(* Logix 5000 project; controller LeakTestAuto vendor 1 type 14 code 226 rev 37.11; software revision 37.01; part 5 of 13 *)
(* tags used below, declared in another part *)
   AOI_Barcode_Comms : AOI_CommStatus;
   AOI_CTS1 : AOI_CTS_INSTRUMENT;
   AOI_CTS1_Comms : AOI_CommStatus;
   AOI_CTS2 : AOI_CTS_INSTRUMENT;
   AOI_CTS2_Comms : AOI_CommStatus;
   AOI_GetShift : AOI_GetShift;
   AOI_RFID_Comms : AOI_CommStatus;
   AOI_Robot_Comms : AOI_CommStatus;
   AOI_RobotPos : AOI_RobotPositions;
   AOI_SeqSteps : AOI_StandardSeqSteps;
   BarcodeScanner : udt_OutputStructure;
   CapActuators_Seq : udt_SequenceStructure_X64;
   CapCTS_Seq : udt_SequenceStructure_X64;
   CapCylinders_Seq : udt_SequenceStructure_X64;
   CapFail_Seq : udt_SequenceStructure_X64;
   CapPass_Seq : udt_SequenceStructure_X64;
   CapRobot_Seq : udt_SequenceStructure_X64;
   CapShuffle_Seq : udt_SequenceStructure_X64;
   Conveyor : udt_OutputStructure;
   ConveyorHomeCounter : COUNTER;
   DryCycle_N1Ready : BOOL;
   DryCycle_N2Ready : BOOL;
   HMI_CloseDisplay : DINT;
   HomingClearNestsBypass : BOOL;
   LastShiftNumber : DINT;
   LeakTester1 : udt_OutputStructure;
   LeakTester2 : udt_OutputStructure;
   Mode_CapActuators : BOOL;
   Mode_CapCTS : BOOL;
   Mode_CapCylinders : BOOL;
   Mode_CapFail : BOOL;
   Mode_CapPass : BOOL;
   Mode_CapRobot : BOOL;
   Mode_CapShuffle : BOOL;
   Nest1Cylinder : udt_OutputStructure;
   Nest2Cylinder : udt_OutputStructure;
   ONS_CapActuators : BOOL;
   ONS_CapCTS : BOOL;
   ONS_CapCylinders : BOOL;
   ONS_CapFail : BOOL;
   ONS_CapPass : BOOL;
   ONS_CapRobot : BOOL;
   ONS_CapShuffle : BOOL;
   ONS_CycleStop : BOOL;
   ONS_ManuMode : BOOL;
   OP220 : udt_Mode;
   OP220_PartToPartCycleTMR : TIMER;
   OP220_Seq : udt_SequenceStructure_X64;
   RFIDScanner : udt_OutputStructure;
   Robot : udt_OutputStructure;
   RobotGripper : udt_OutputStructure;
   RobotInputs : udt_EpsonInputs;
   RobotOutputs : udt_EpsonOutputs;
   ShiftTimes : SINT[24];
   TON_HMICloseDisplayDelay : TIMER;
   ConveyorPurgeCounter : DINT;   // Outfeed Coveyor Purge Counter
   DateString : String20;
   DateTimeString : String20;
   HMI_PurgeCycleSP : DINT;   // HMI Purge Cycles Setpoint
   I_OP220_N3_CONVEYOR_CLEAT : ALIAS FOR Local:3:I.Pt13.Data;
   I_OP220_N3_CONVEYOR_LOAD : ALIAS FOR Local:3:I.Pt12.Data;
   I_OP220_N3_CONVEYOR_UNLOAD : ALIAS FOR Local:3:I.Pt14.Data;
   I_OP220_N3_DUT_PRE_NEST_0 : ALIAS FOR Local:3:I.Pt00.Data;
   I_OP220_N3_DUT_PRE_NEST_1 : ALIAS FOR Local:3:I.Pt01.Data;
   I_OP220_N3_DUT_PRE_NEST_2 : ALIAS FOR Local:3:I.Pt02.Data;
   I_OP220_N3_MAIN_AIR_OK : ALIAS FOR Local:3:I.Pt07.Data;
   I_OP220_N3_NEST1_EXTEND : ALIAS FOR Local:3:I.Pt04.Data;
   I_OP220_N3_NEST1_HOME : ALIAS FOR Local:3:I.Pt03.Data;
   I_OP220_N3_NEST2_EXTEND : ALIAS FOR Local:3:I.Pt06.Data;
   I_OP220_N3_NEST2_HOME : ALIAS FOR Local:3:I.Pt05.Data;
   I_OP220_N3_REJECT_BIN_OK : ALIAS FOR Local:3:I.Pt09.Data;
   IOCounterHasRef : BOOL;
   IOTriggerCounts : UDINT[128];
   James_Dint : DINT;   // James Test Word
   LastPLCEdit : String20;
   LastPLCEditHistory : String20[20];
   O_OP220_N5_EN_LT_BU : ALIAS FOR Local:5:O.Pt03.Data;
   O_OP220_N5_EN_LT_GN : ALIAS FOR Local:5:O.Pt00.Data;
   O_OP220_N5_EN_LT_RD : ALIAS FOR Local:5:O.Pt02.Data;
   O_OP220_N5_EN_LT_YE : ALIAS FOR Local:5:O.Pt01.Data;
   OP220_ConsumedFromMain_PurgeModeEn : BOOL;
   OP220_Power : BOOL;
   PLC : AOI_PLC;
   Purge_Count_DN : BOOL;   // Purge Counter Completed
   ShiftChange : BOOL;
   ShiftNumber : SINT;
   TimeString : String20;
   TON_PLC_BootUp : TIMER;
(* MainProgram, continued *)

ROUTINE AManualDebug   (* ladder *)
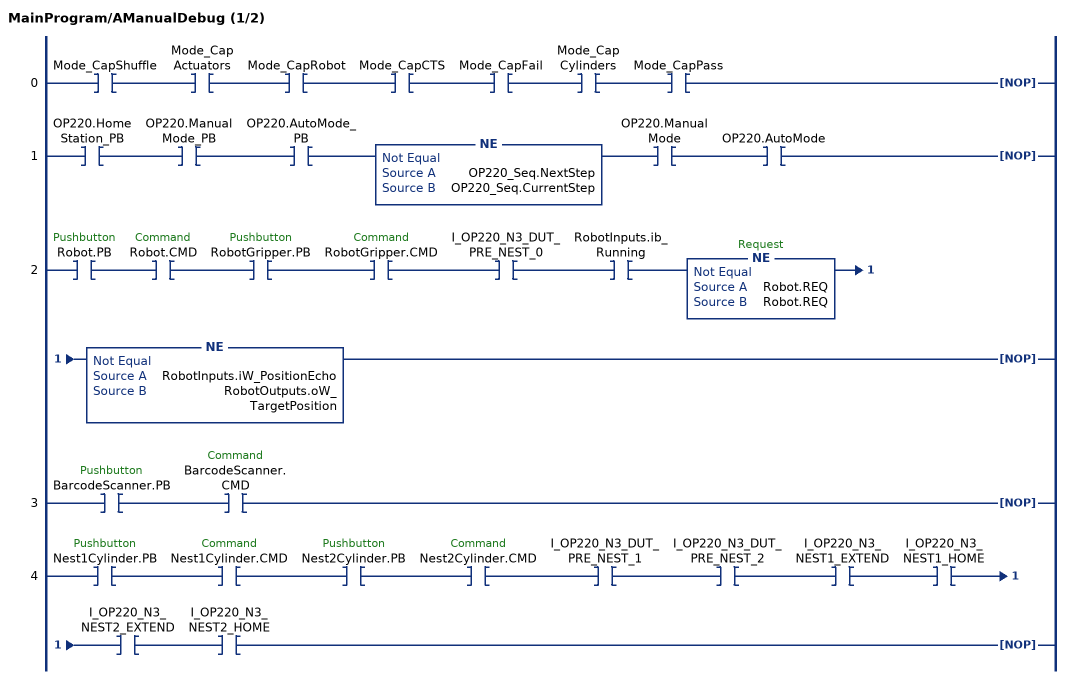
   0: XIC(Mode_CapShuffle)XIC(Mode_CapActuators)XIC(Mode_CapRobot)XIC(Mode_CapCTS)XIC(Mode_CapFail)XIC(Mode_CapCylinders)XIC(Mode_CapPass)NOP();
   1: XIC(OP220.HomeStation_PB)XIC(OP220.ManualMode_PB)XIC(OP220.AutoMode_PB)NE(OP220_Seq.NextStep,OP220_Seq.CurrentStep)XIC(OP220.ManualMode)XIC(OP220.AutoMode)NOP();
   2: XIC(Robot.PB)XIC(Robot.CMD)XIC(RobotGripper.PB)XIC(RobotGripper.CMD)XIC(I_OP220_N3_DUT_PRE_NEST_0)XIC(RobotInputs.ib_Running)NE(Robot.REQ,Robot.REQ)NE(RobotInputs.iW_PositionEcho,RobotOutputs.oW_TargetPosition)NOP();
   3: XIC(BarcodeScanner.PB)XIC(BarcodeScanner.CMD)NOP();
   4: XIC(Nest1Cylinder.PB)XIC(Nest1Cylinder.CMD)XIC(Nest2Cylinder.PB)XIC(Nest2Cylinder.CMD)XIC(I_OP220_N3_DUT_PRE_NEST_1)XIC(I_OP220_N3_DUT_PRE_NEST_2)XIC(I_OP220_N3_NEST1_EXTEND)XIC(I_OP220_N3_NEST1_HOME)XIC(I_OP220_N3_NEST2_EXTEND)XIC(I_OP220_N3_NEST2_HOME)NOP();
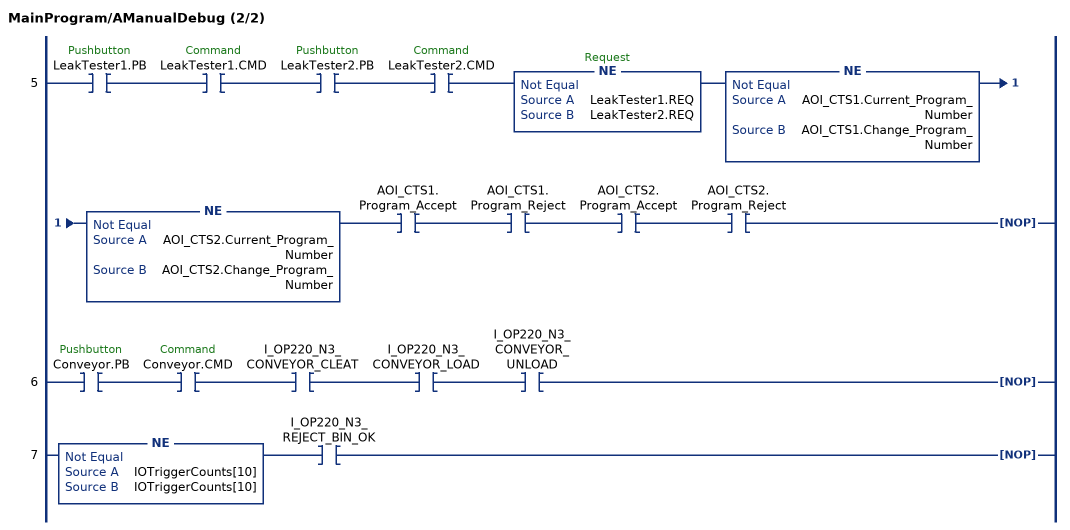
   5: XIC(LeakTester1.PB)XIC(LeakTester1.CMD)XIC(LeakTester2.PB)XIC(LeakTester2.CMD)NE(LeakTester1.REQ,LeakTester2.REQ)NE(AOI_CTS1.Current_Program_Number,AOI_CTS1.Change_Program_Number)NE(AOI_CTS2.Current_Program_Number,AOI_CTS2.Change_Program_Number)XIC(AOI_CTS1.Program_Accept)XIC(AOI_CTS1.Program_Reject)XIC(AOI_CTS2.Program_Accept)XIC(AOI_CTS2.Program_Reject)NOP();
   6: XIC(Conveyor.PB)XIC(Conveyor.CMD)XIC(I_OP220_N3_CONVEYOR_CLEAT)XIC(I_OP220_N3_CONVEYOR_LOAD)XIC(I_OP220_N3_CONVEYOR_UNLOAD)NOP();
   7: NE(IOTriggerCounts[10],IOTriggerCounts[10])XIC(I_OP220_N3_REJECT_BIN_OK)NOP();
END_ROUTINE

ROUTINE MainRoutine   (* ladder *)
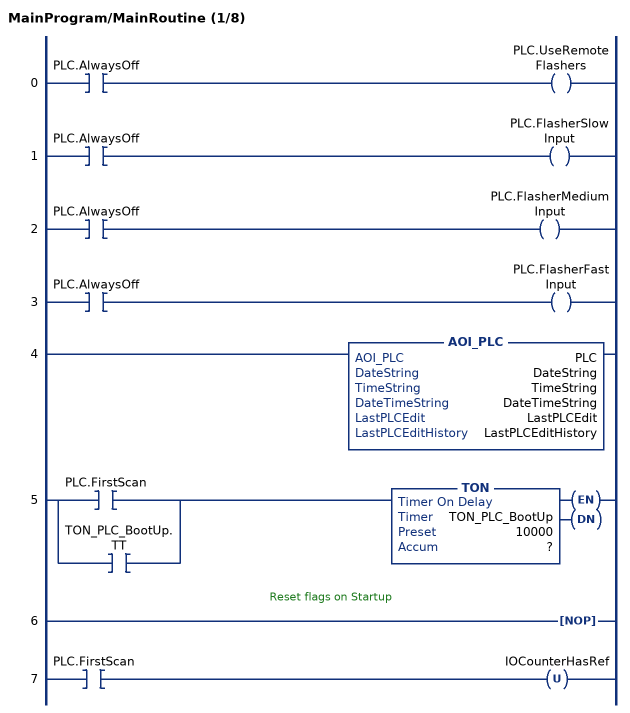
   0: XIC(PLC.AlwaysOff)OTE(PLC.UseRemoteFlashers);
   1: XIC(PLC.AlwaysOff)OTE(PLC.FlasherSlowInput);
   2: XIC(PLC.AlwaysOff)OTE(PLC.FlasherMediumInput);
   3: XIC(PLC.AlwaysOff)OTE(PLC.FlasherFastInput);
   4: AOI_PLC(PLC,DateString,TimeString,DateTimeString,LastPLCEdit,LastPLCEditHistory);
   5: [XIC(PLC.FirstScan) ,XIC(TON_PLC_BootUp.TT) ]TON(TON_PLC_BootUp,?,?);
   // Reset flags on Startup
   6: NOP();
   7: XIC(PLC.FirstScan)OTU(IOCounterHasRef);
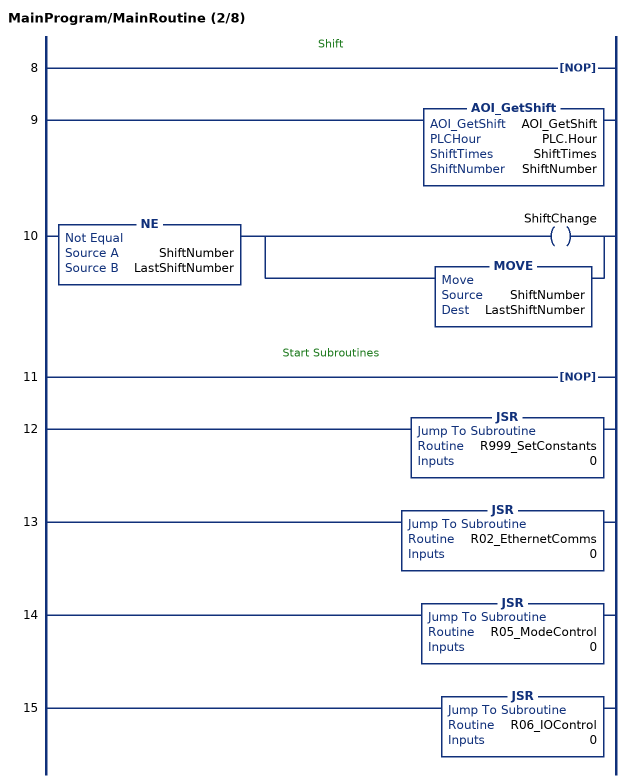
   // Shift
   8: NOP();
   9: AOI_GetShift(AOI_GetShift,PLC.Hour,ShiftTimes,ShiftNumber);
   10: NE(ShiftNumber,LastShiftNumber)[OTE(ShiftChange) ,MOVE(ShiftNumber,LastShiftNumber) ];
   // Start Subroutines
   11: NOP();
   12: JSR(R999_SetConstants,0);
   13: JSR(R02_EthernetComms,0);
   14: JSR(R05_ModeControl,0);
   15: JSR(R06_IOControl,0);
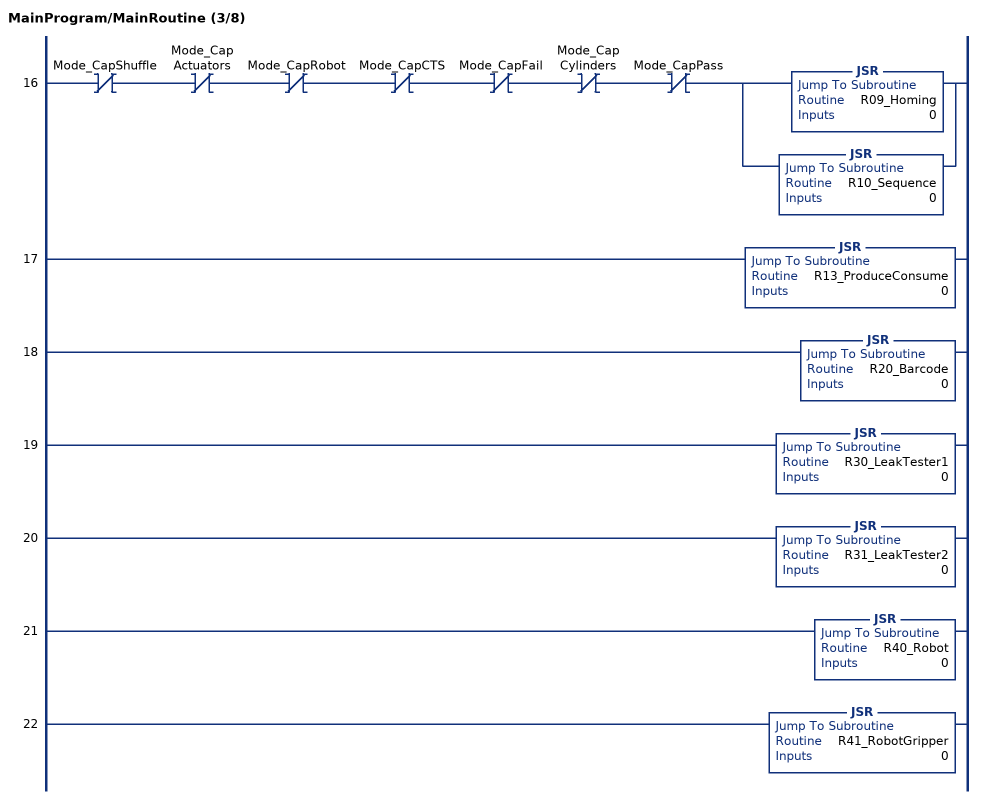
   16: XIO(Mode_CapShuffle)XIO(Mode_CapActuators)XIO(Mode_CapRobot)XIO(Mode_CapCTS)XIO(Mode_CapFail)XIO(Mode_CapCylinders)XIO(Mode_CapPass)[JSR(R09_Homing,0) ,JSR(R10_Sequence,0) ];
   17: JSR(R13_ProduceConsume,0);
   18: JSR(R20_Barcode,0);
   19: JSR(R30_LeakTester1,0);
   20: JSR(R31_LeakTester2,0);
   21: JSR(R40_Robot,0);
   22: JSR(R41_RobotGripper,0);
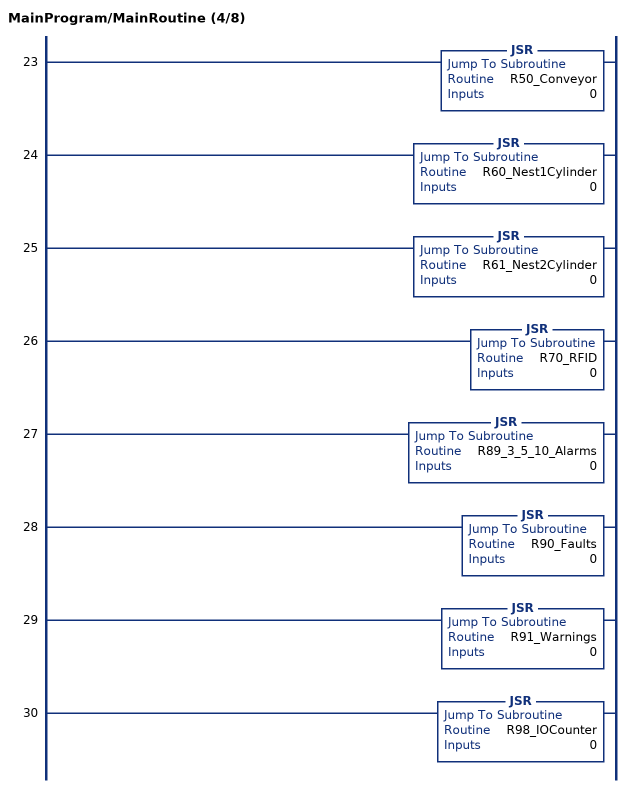
   23: JSR(R50_Conveyor,0);
   24: JSR(R60_Nest1Cylinder,0);
   25: JSR(R61_Nest2Cylinder,0);
   26: JSR(R70_RFID,0);
   27: JSR(R89_3_5_10_Alarms,0);
   28: JSR(R90_Faults,0);
   29: JSR(R91_Warnings,0);
   30: JSR(R98_IOCounter,0);
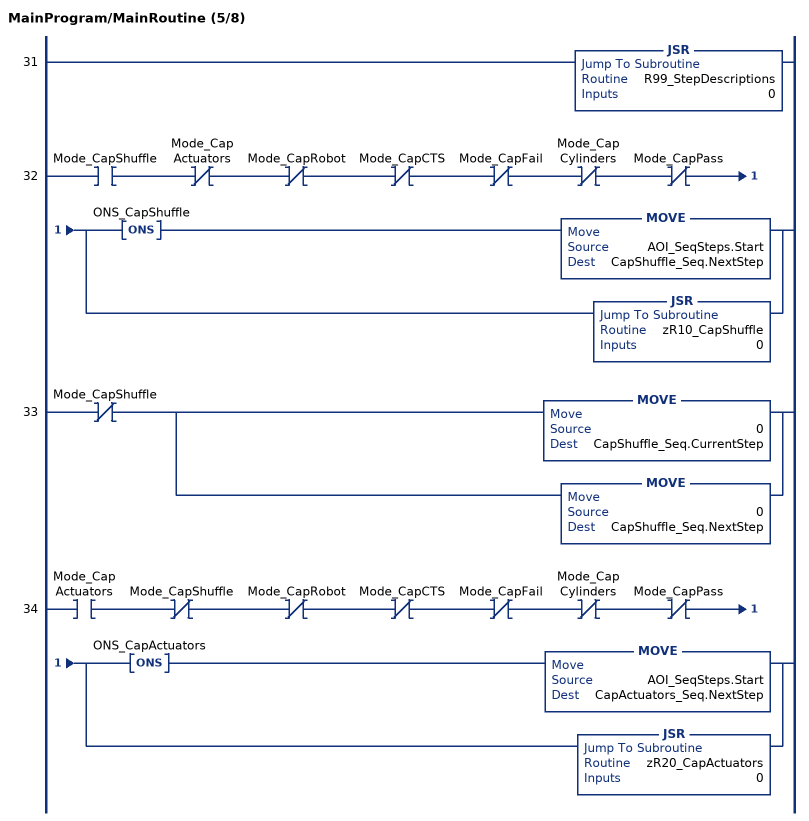
   31: JSR(R99_StepDescriptions,0);
   32: XIC(Mode_CapShuffle)XIO(Mode_CapActuators)XIO(Mode_CapRobot)XIO(Mode_CapCTS)XIO(Mode_CapFail)XIO(Mode_CapCylinders)XIO(Mode_CapPass)[ONS(ONS_CapShuffle) MOVE(AOI_SeqSteps.Start,CapShuffle_Seq.NextStep) ,JSR(zR10_CapShuffle,0) ];
   33: XIO(Mode_CapShuffle)[MOVE(0,CapShuffle_Seq.CurrentStep) ,MOVE(0,CapShuffle_Seq.NextStep) ];
   34: XIC(Mode_CapActuators)XIO(Mode_CapShuffle)XIO(Mode_CapRobot)XIO(Mode_CapCTS)XIO(Mode_CapFail)XIO(Mode_CapCylinders)XIO(Mode_CapPass)[ONS(ONS_CapActuators) MOVE(AOI_SeqSteps.Start,CapActuators_Seq.NextStep) ,JSR(zR20_CapActuators,0) ];
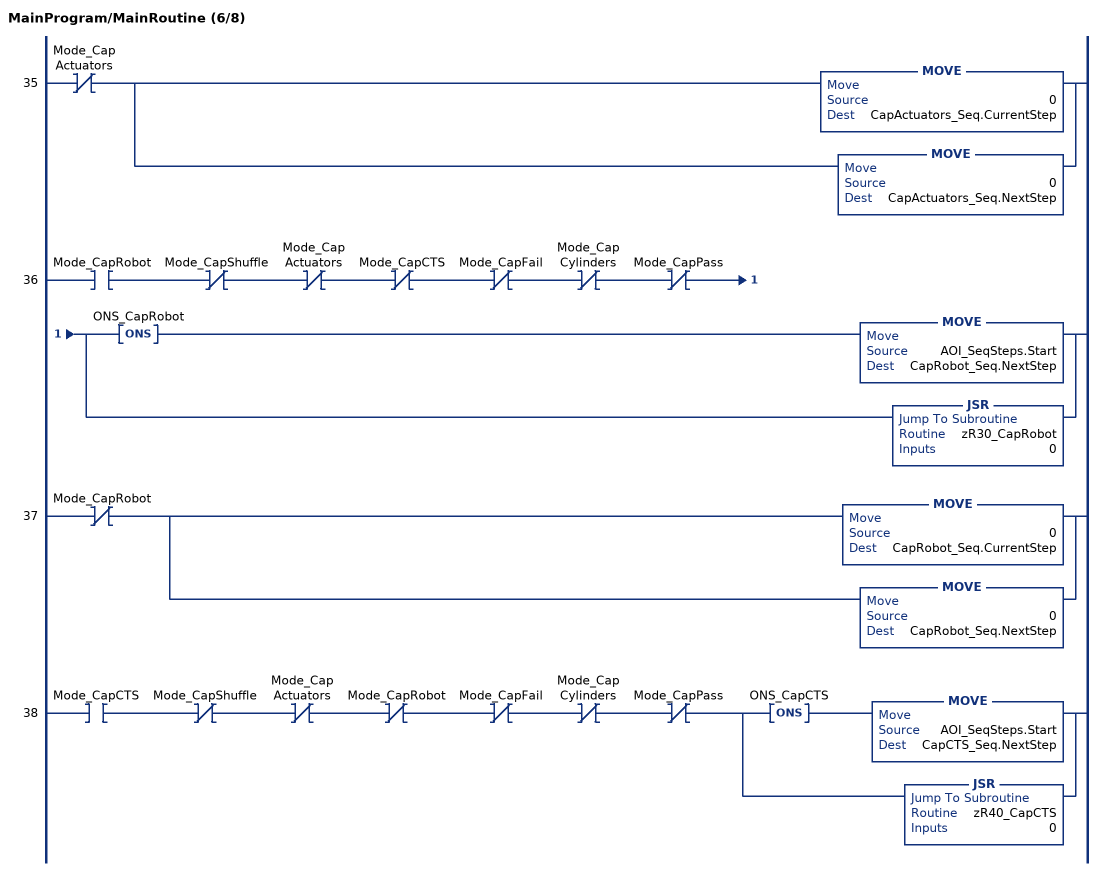
   35: XIO(Mode_CapActuators)[MOVE(0,CapActuators_Seq.CurrentStep) ,MOVE(0,CapActuators_Seq.NextStep) ];
   36: XIC(Mode_CapRobot)XIO(Mode_CapShuffle)XIO(Mode_CapActuators)XIO(Mode_CapCTS)XIO(Mode_CapFail)XIO(Mode_CapCylinders)XIO(Mode_CapPass)[ONS(ONS_CapRobot) MOVE(AOI_SeqSteps.Start,CapRobot_Seq.NextStep) ,JSR(zR30_CapRobot,0) ];
   37: XIO(Mode_CapRobot)[MOVE(0,CapRobot_Seq.CurrentStep) ,MOVE(0,CapRobot_Seq.NextStep) ];
   38: XIC(Mode_CapCTS)XIO(Mode_CapShuffle)XIO(Mode_CapActuators)XIO(Mode_CapRobot)XIO(Mode_CapFail)XIO(Mode_CapCylinders)XIO(Mode_CapPass)[ONS(ONS_CapCTS) MOVE(AOI_SeqSteps.Start,CapCTS_Seq.NextStep) ,JSR(zR40_CapCTS,0) ];
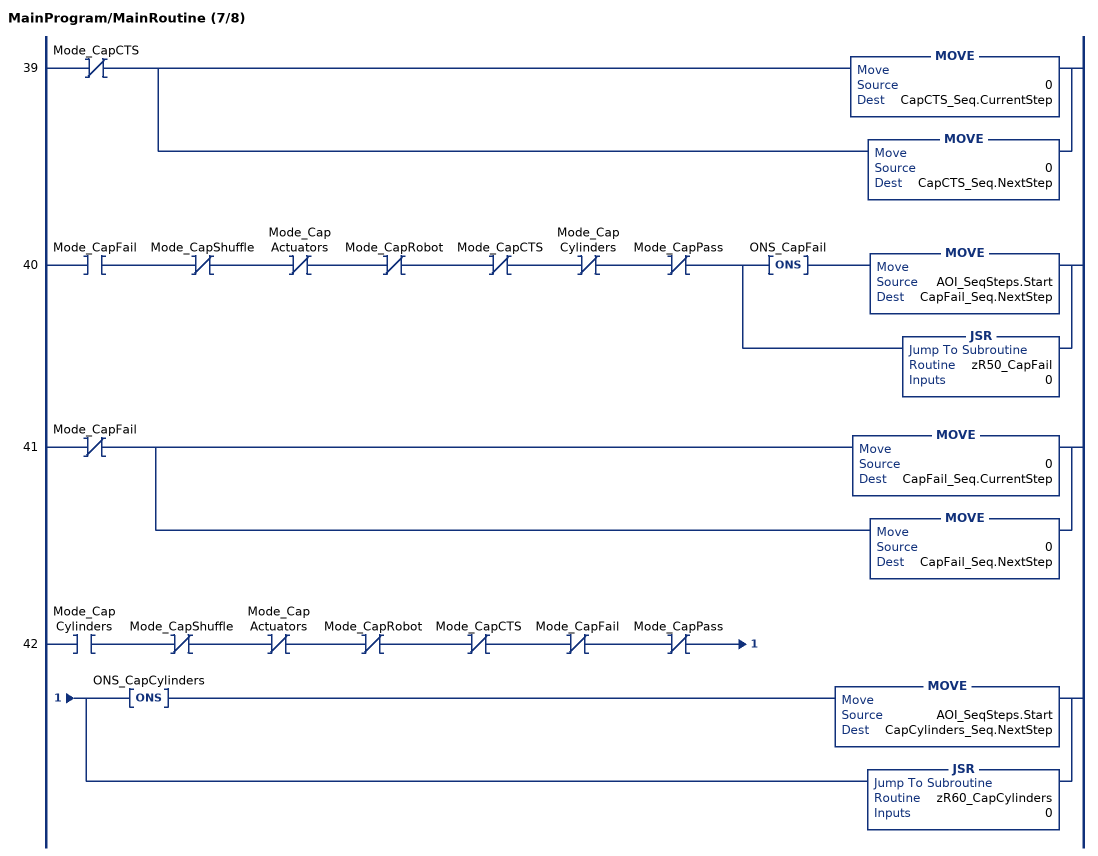
   39: XIO(Mode_CapCTS)[MOVE(0,CapCTS_Seq.CurrentStep) ,MOVE(0,CapCTS_Seq.NextStep) ];
   40: XIC(Mode_CapFail)XIO(Mode_CapShuffle)XIO(Mode_CapActuators)XIO(Mode_CapRobot)XIO(Mode_CapCTS)XIO(Mode_CapCylinders)XIO(Mode_CapPass)[ONS(ONS_CapFail) MOVE(AOI_SeqSteps.Start,CapFail_Seq.NextStep) ,JSR(zR50_CapFail,0) ];
   41: XIO(Mode_CapFail)[MOVE(0,CapFail_Seq.CurrentStep) ,MOVE(0,CapFail_Seq.NextStep) ];
   42: XIC(Mode_CapCylinders)XIO(Mode_CapShuffle)XIO(Mode_CapActuators)XIO(Mode_CapRobot)XIO(Mode_CapCTS)XIO(Mode_CapFail)XIO(Mode_CapPass)[ONS(ONS_CapCylinders) MOVE(AOI_SeqSteps.Start,CapCylinders_Seq.NextStep) ,JSR(zR60_CapCylinders,0) ];
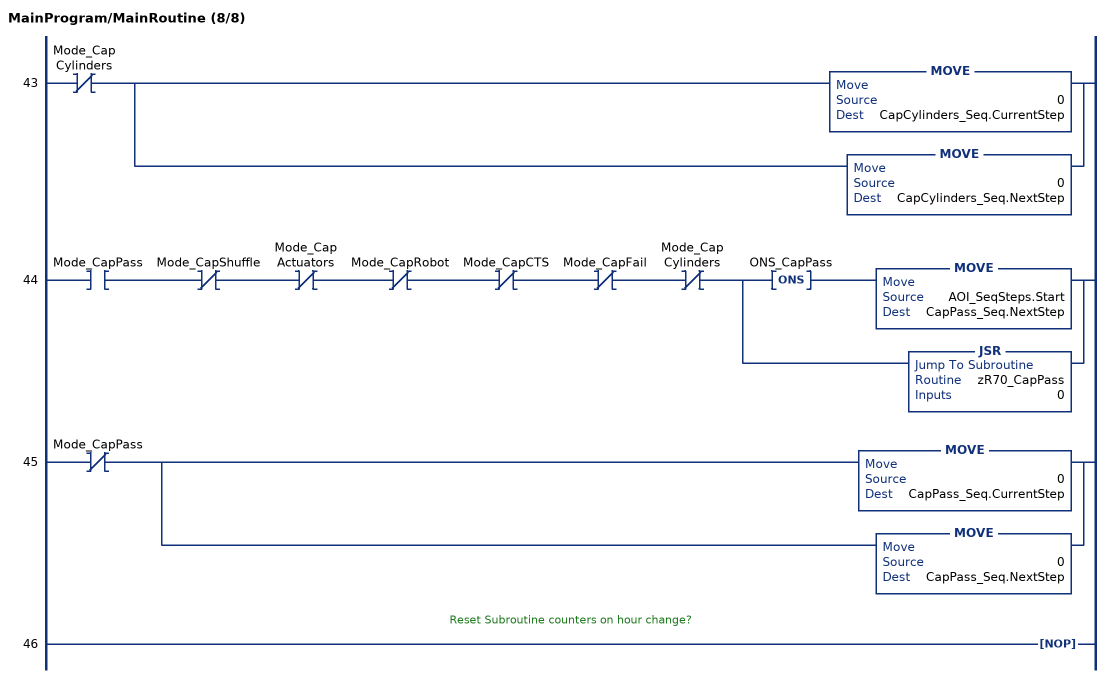
   43: XIO(Mode_CapCylinders)[MOVE(0,CapCylinders_Seq.CurrentStep) ,MOVE(0,CapCylinders_Seq.NextStep) ];
   44: XIC(Mode_CapPass)XIO(Mode_CapShuffle)XIO(Mode_CapActuators)XIO(Mode_CapRobot)XIO(Mode_CapCTS)XIO(Mode_CapFail)XIO(Mode_CapCylinders)[ONS(ONS_CapPass) MOVE(AOI_SeqSteps.Start,CapPass_Seq.NextStep) ,JSR(zR70_CapPass,0) ];
   45: XIO(Mode_CapPass)[MOVE(0,CapPass_Seq.CurrentStep) ,MOVE(0,CapPass_Seq.NextStep) ];
   // Reset Subroutine counters on hour change?
   46: NOP();
END_ROUTINE

ROUTINE R02_EthernetComms   (* ladder *)
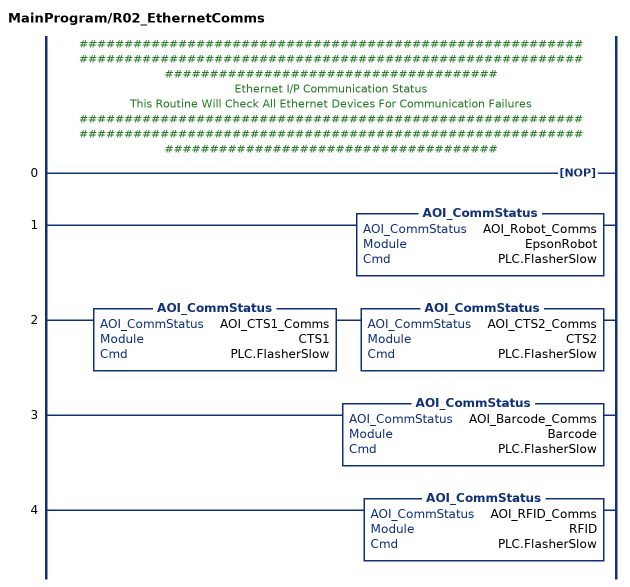
   // #####################################################################################################################################################
   // Ethernet I/P Communication Status
   // This Routine Will Check All Ethernet Devices For Communication Failures
   // #####################################################################################################################################################
   0: NOP();
   1: AOI_CommStatus(AOI_Robot_Comms,EpsonRobot,PLC.FlasherSlow);
   2: AOI_CommStatus(AOI_CTS1_Comms,CTS1,PLC.FlasherSlow)AOI_CommStatus(AOI_CTS2_Comms,CTS2,PLC.FlasherSlow);
   3: AOI_CommStatus(AOI_Barcode_Comms,Barcode,PLC.FlasherSlow);
   4: AOI_CommStatus(AOI_RFID_Comms,RFID,PLC.FlasherSlow);
END_ROUTINE

ROUTINE R05_ModeControl   (* ladder *)
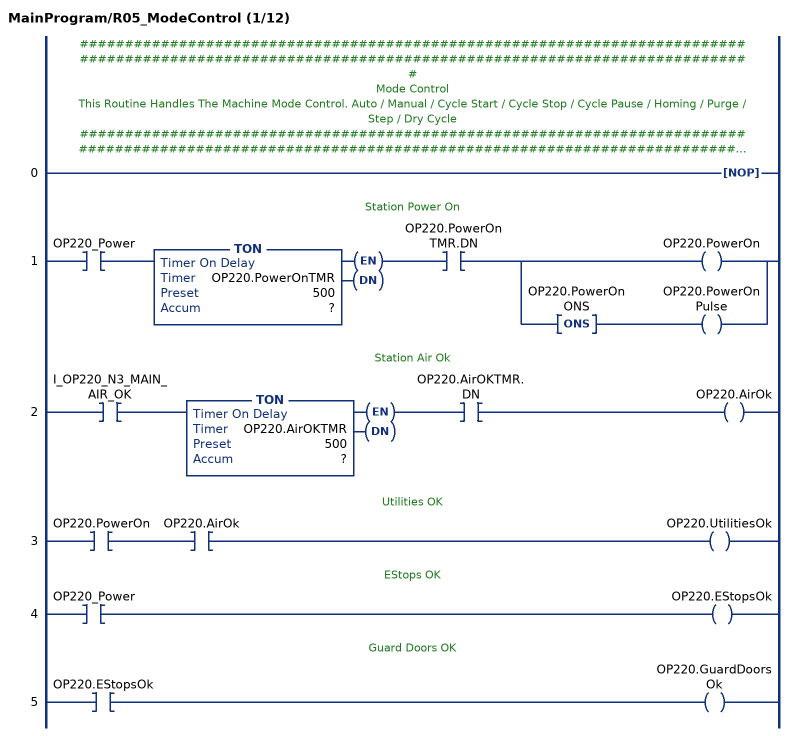
   // #####################################################################################################################################################
   // Mode Control
   // This Routine Handles The Machine Mode Control. Auto / Manual / Cycle Start / Cycle Stop / Cycle Pause / Homing / Purge / Step / Dry Cycle
   // #####################################################################################################################################################
   0: NOP();
   // Station Power On
   1: XIC(OP220_Power)TON(OP220.PowerOnTMR,?,?)XIC(OP220.PowerOnTMR.DN)[OTE(OP220.PowerOn) ,ONS(OP220.PowerOnONS) OTE(OP220.PowerOnPulse) ];
   // Station Air Ok
   2: XIC(I_OP220_N3_MAIN_AIR_OK)TON(OP220.AirOKTMR,?,?)XIC(OP220.AirOKTMR.DN)OTE(OP220.AirOk);
   // Utilities OK
   3: XIC(OP220.PowerOn)XIC(OP220.AirOk)OTE(OP220.UtilitiesOk);
   // EStops OK
   4: XIC(OP220_Power)OTE(OP220.EStopsOk);
   // Guard Doors OK
   5: XIC(OP220.EStopsOk)OTE(OP220.GuardDoorsOk);
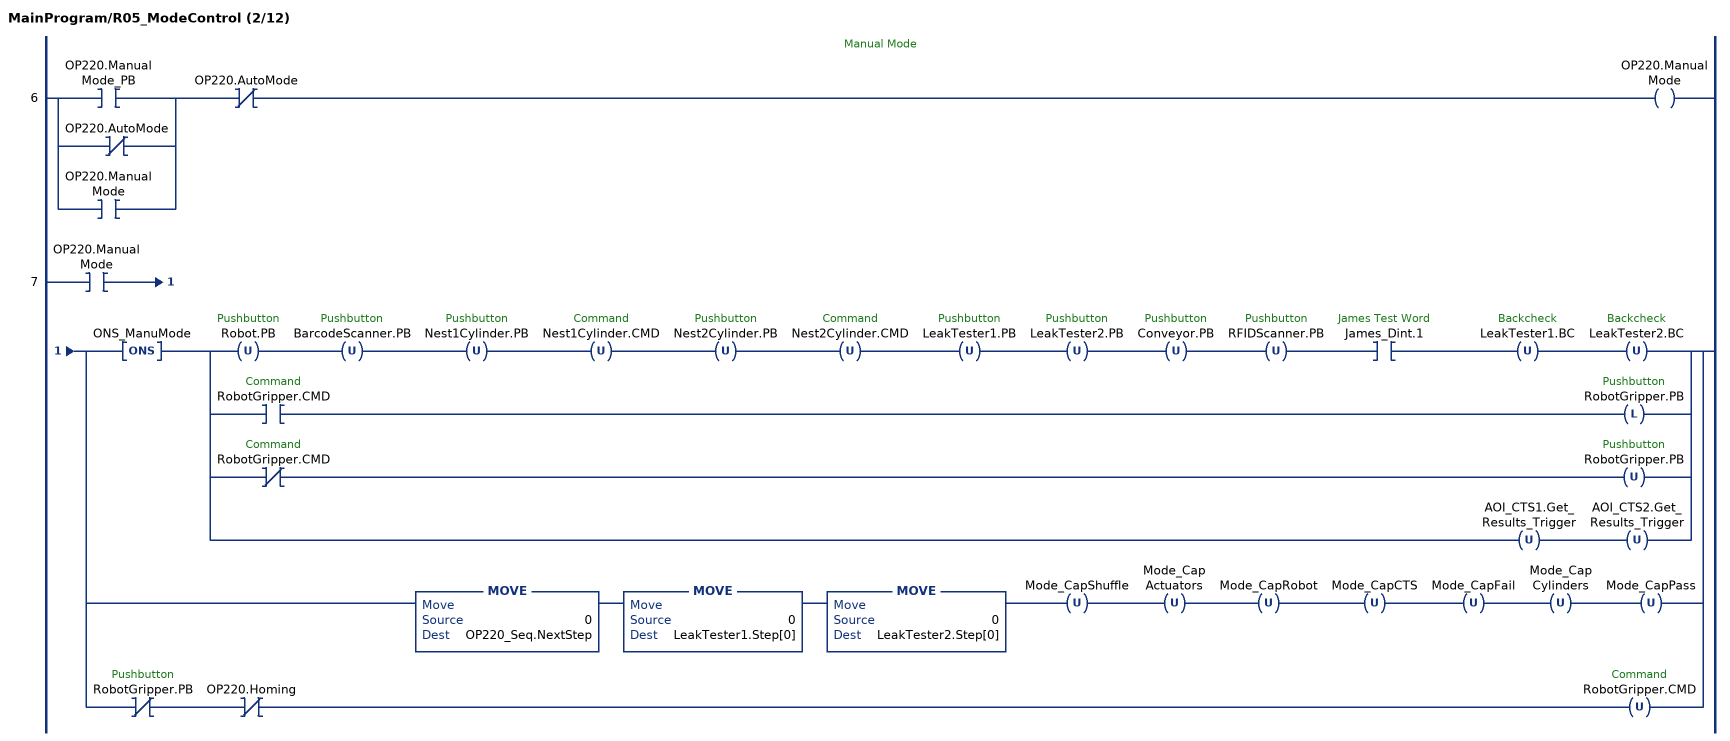
   // Manual Mode
   6: [XIC(OP220.ManualMode_PB) ,XIO(OP220.AutoMode) ,XIC(OP220.ManualMode) ]XIO(OP220.AutoMode)OTE(OP220.ManualMode);
   7: XIC(OP220.ManualMode)[ONS(ONS_ManuMode) [OTU(Robot.PB) OTU(BarcodeScanner.PB) OTU(Nest1Cylinder.PB) OTU(Nest1Cylinder.CMD) OTU(Nest2Cylinder.PB) OTU(Nest2Cylinder.CMD) OTU(LeakTester1.PB) OTU(LeakTester2.PB) OTU(Conveyor.PB) OTU(RFIDScanner.PB) XIC(James_Dint.1) OTU(LeakTester1.BC) OTU(LeakTester2.BC) ,XIC(RobotGripper.CMD) OTL(RobotGripper.PB) ,XIO(RobotGripper.CMD) OTU(RobotGripper.PB) ,OTU(AOI_CTS1.Get_Results_Trigger) OTU(AOI_CTS2.Get_Results_Trigger) ] ,MOVE(0,OP220_Seq.NextStep) MOVE(0,LeakTester1.Step[0]) MOVE(0,LeakTester2.Step[0]) OTU(Mode_CapShuffle) OTU(Mode_CapActuators) OTU(Mode_CapRobot) OTU(Mode_CapCTS) OTU(Mode_CapFail) OTU(Mode_CapCylinders) OTU(Mode_CapPass) ,XIO(RobotGripper.PB) XIO(OP220.Homing) OTU(RobotGripper.CMD) ];
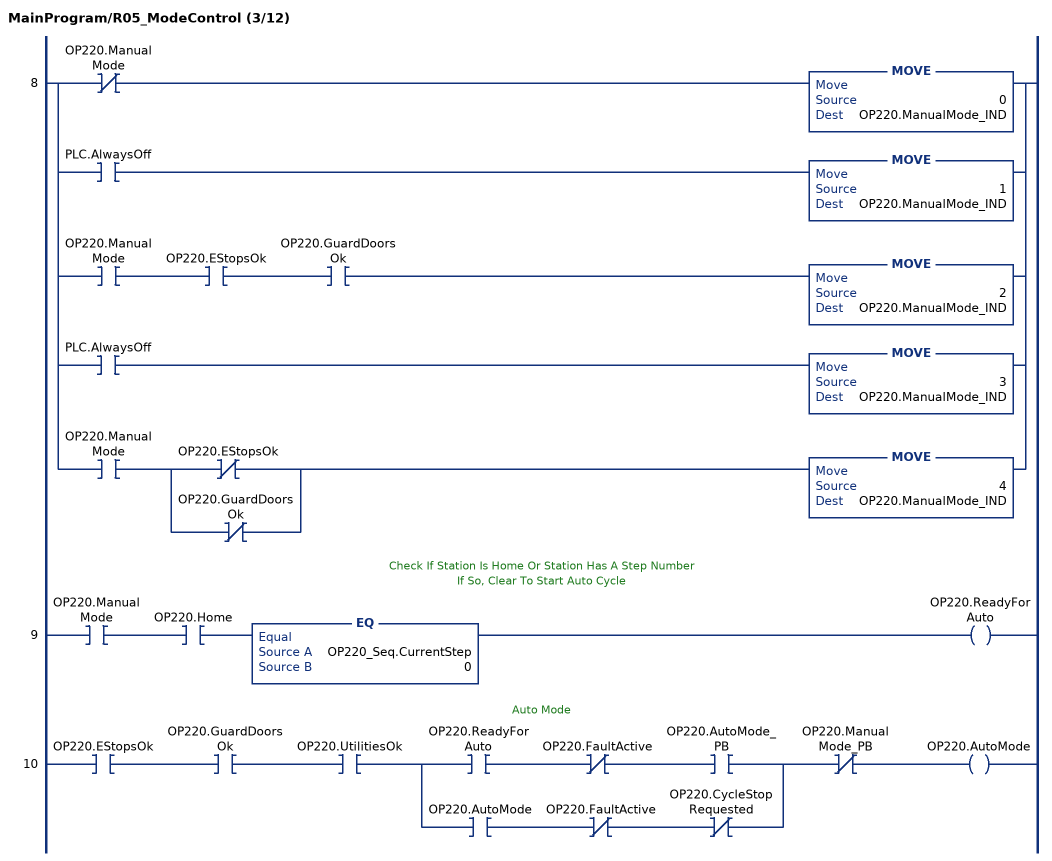
   8: [XIO(OP220.ManualMode) MOVE(0,OP220.ManualMode_IND) ,XIC(PLC.AlwaysOff) MOVE(1,OP220.ManualMode_IND) ,XIC(OP220.ManualMode) XIC(OP220.EStopsOk) XIC(OP220.GuardDoorsOk) MOVE(2,OP220.ManualMode_IND) ,XIC(PLC.AlwaysOff) MOVE(3,OP220.ManualMode_IND) ,XIC(OP220.ManualMode) [XIO(OP220.EStopsOk) ,XIO(OP220.GuardDoorsOk) ] MOVE(4,OP220.ManualMode_IND) ];
   // Check If Station Is Home Or Station Has A Step Number
   // If So, Clear To Start Auto Cycle
   9: XIC(OP220.ManualMode)XIC(OP220.Home)EQ(OP220_Seq.CurrentStep,0)OTE(OP220.ReadyForAuto);
   // Auto Mode
   10: XIC(OP220.EStopsOk)XIC(OP220.GuardDoorsOk)XIC(OP220.UtilitiesOk)[XIC(OP220.ReadyForAuto) XIO(OP220.FaultActive) XIC(OP220.AutoMode_PB) ,XIC(OP220.AutoMode) XIO(OP220.FaultActive) XIO(OP220.CycleStopRequested) ]XIO(OP220.ManualMode_PB)OTE(OP220.AutoMode);
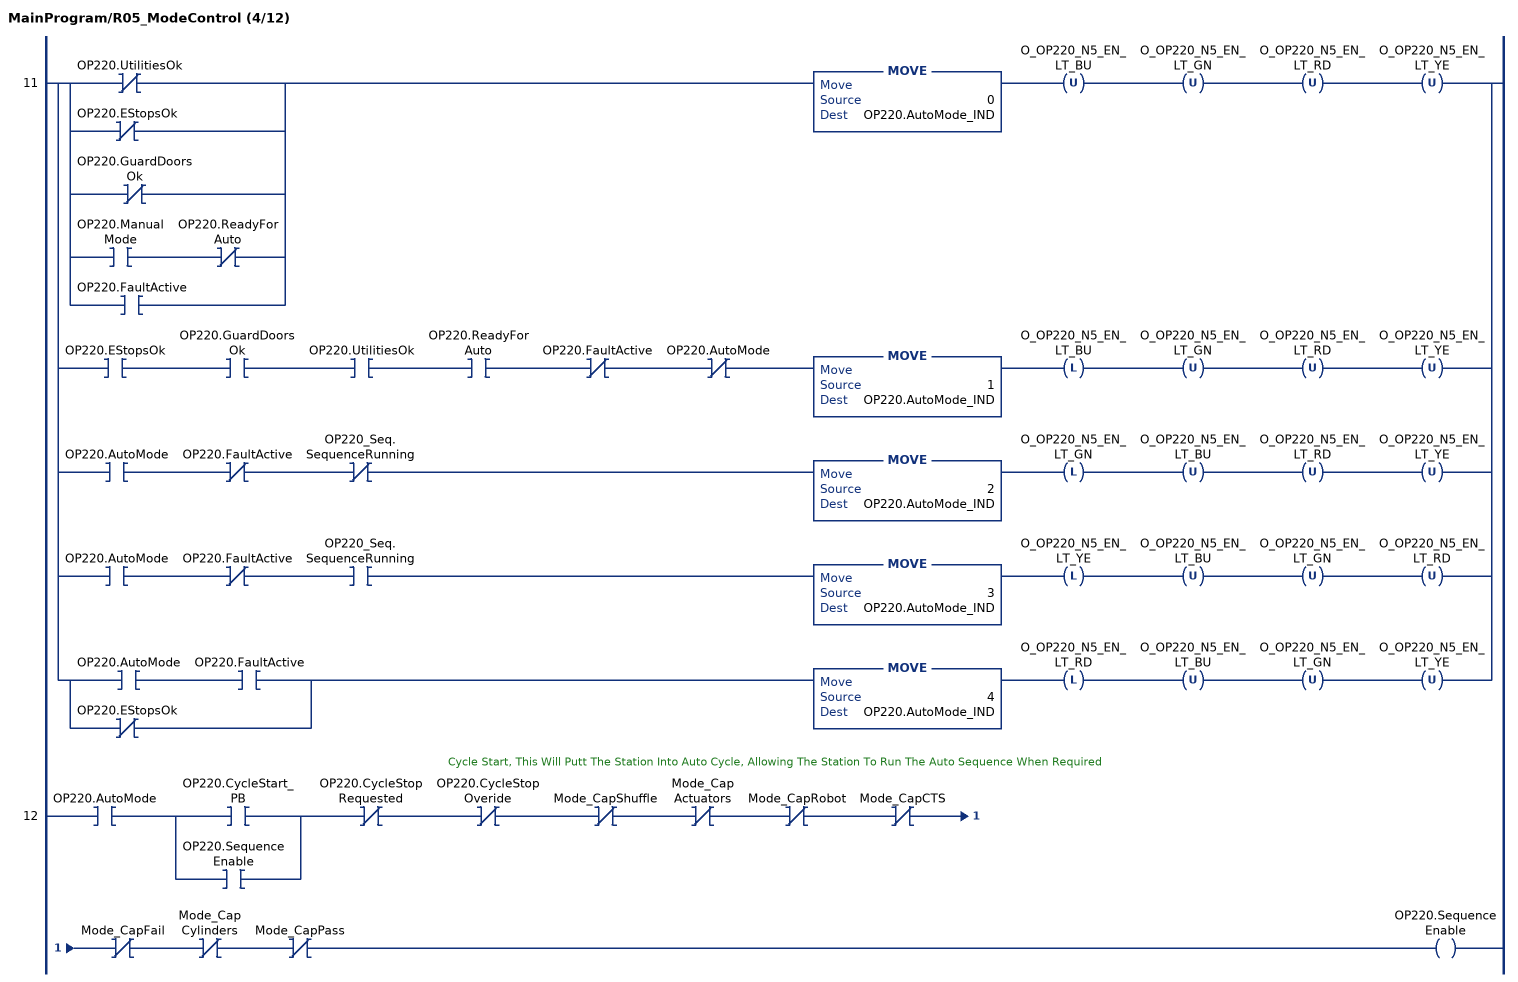
   11: [[XIO(OP220.UtilitiesOk) ,XIO(OP220.EStopsOk) ,XIO(OP220.GuardDoorsOk) ,XIC(OP220.ManualMode) XIO(OP220.ReadyForAuto) ,XIC(OP220.FaultActive) ] MOVE(0,OP220.AutoMode_IND) OTU(O_OP220_N5_EN_LT_BU) OTU(O_OP220_N5_EN_LT_GN) OTU(O_OP220_N5_EN_LT_RD) OTU(O_OP220_N5_EN_LT_YE) ,XIC(OP220.EStopsOk) XIC(OP220.GuardDoorsOk) XIC(OP220.UtilitiesOk) XIC(OP220.ReadyForAuto) XIO(OP220.FaultActive) XIO(OP220.AutoMode) MOVE(1,OP220.AutoMode_IND) OTL(O_OP220_N5_EN_LT_BU) OTU(O_OP220_N5_EN_LT_GN) OTU(O_OP220_N5_EN_LT_RD) OTU(O_OP220_N5_EN_LT_YE) ,XIC(OP220.AutoMode) XIO(OP220.FaultActive) XIO(OP220_Seq.SequenceRunning) MOVE(2,OP220.AutoMode_IND) OTL(O_OP220_N5_EN_LT_GN) OTU(O_OP220_N5_EN_LT_BU) OTU(O_OP220_N5_EN_LT_RD) OTU(O_OP220_N5_EN_LT_YE) ,XIC(OP220.AutoMode) XIO(OP220.FaultActive) XIC(OP220_Seq.SequenceRunning) MOVE(3,OP220.AutoMode_IND) OTL(O_OP220_N5_EN_LT_YE) OTU(O_OP220_N5_EN_LT_BU) OTU(O_OP220_N5_EN_LT_GN) OTU(O_OP220_N5_EN_LT_RD) ,[XIC(OP220.AutoMode) XIC(OP220.FaultActive) ,XIO(OP220.EStopsOk) ] MOVE(4,OP220.AutoMode_IND) OTL(O_OP220_N5_EN_LT_RD) OTU(O_OP220_N5_EN_LT_BU) OTU(O_OP220_N5_EN_LT_GN) OTU(O_OP220_N5_EN_LT_YE) ];
   // Cycle Start, This Will Putt The Station Into Auto Cycle, Allowing The Station To Run The Auto Sequence When Required
   12: XIC(OP220.AutoMode)[XIC(OP220.CycleStart_PB) ,XIC(OP220.SequenceEnable) ]XIO(OP220.CycleStopRequested)XIO(OP220.CycleStopOveride)XIO(Mode_CapShuffle)XIO(Mode_CapActuators)XIO(Mode_CapRobot)XIO(Mode_CapCTS)XIO(Mode_CapFail)XIO(Mode_CapCylinders)XIO(Mode_CapPass)OTE(OP220.SequenceEnable);
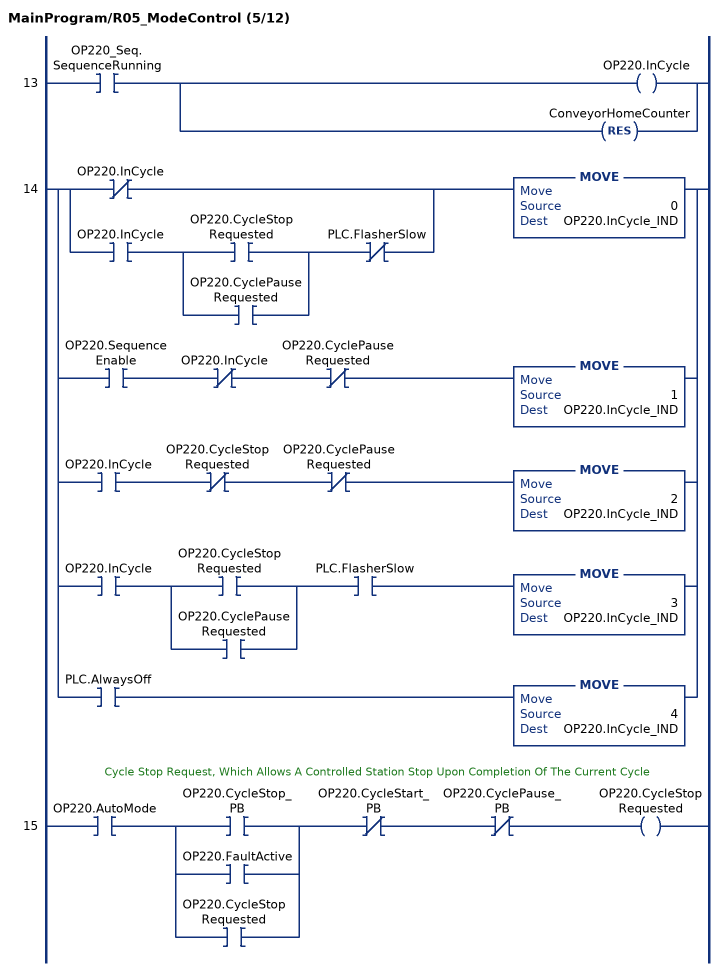
   13: XIC(OP220_Seq.SequenceRunning)[OTE(OP220.InCycle) ,RES(ConveyorHomeCounter) ];
   14: [[XIO(OP220.InCycle) ,XIC(OP220.InCycle) [XIC(OP220.CycleStopRequested) ,XIC(OP220.CyclePauseRequested) ] XIO(PLC.FlasherSlow) ] MOVE(0,OP220.InCycle_IND) ,XIC(OP220.SequenceEnable) XIO(OP220.InCycle) XIO(OP220.CyclePauseRequested) MOVE(1,OP220.InCycle_IND) ,XIC(OP220.InCycle) XIO(OP220.CycleStopRequested) XIO(OP220.CyclePauseRequested) MOVE(2,OP220.InCycle_IND) ,XIC(OP220.InCycle) [XIC(OP220.CycleStopRequested) ,XIC(OP220.CyclePauseRequested) ] XIC(PLC.FlasherSlow) MOVE(3,OP220.InCycle_IND) ,XIC(PLC.AlwaysOff) MOVE(4,OP220.InCycle_IND) ];
   // Cycle Stop Request, Which Allows A Controlled Station Stop Upon Completion Of The Current Cycle
   15: XIC(OP220.AutoMode)[XIC(OP220.CycleStop_PB) ,XIC(OP220.FaultActive) ,XIC(OP220.CycleStopRequested) ]XIO(OP220.CycleStart_PB)XIO(OP220.CyclePause_PB)OTE(OP220.CycleStopRequested);
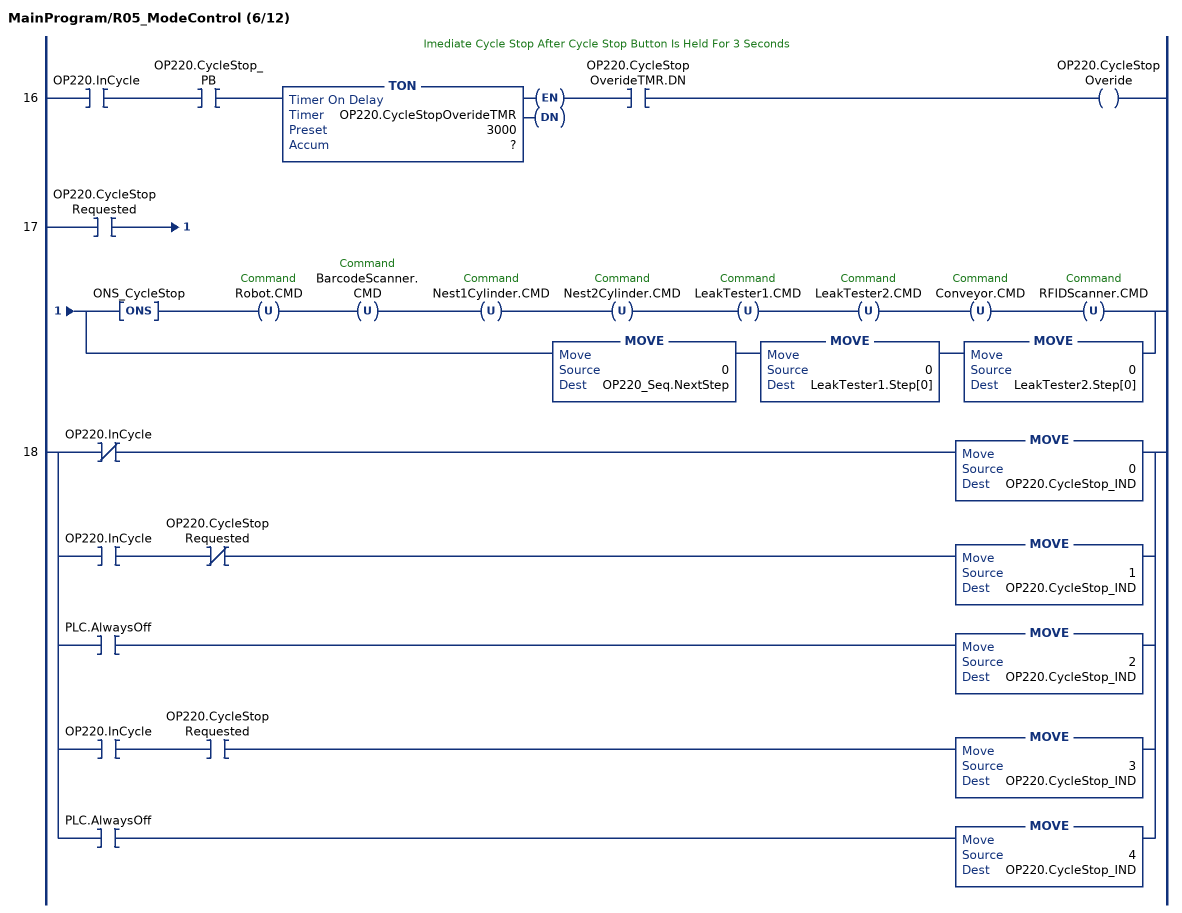
   // Imediate Cycle Stop After Cycle Stop Button Is Held For 3 Seconds
   16: XIC(OP220.InCycle)XIC(OP220.CycleStop_PB)TON(OP220.CycleStopOverideTMR,?,?)XIC(OP220.CycleStopOverideTMR.DN)OTE(OP220.CycleStopOveride);
   17: XIC(OP220.CycleStopRequested)[ONS(ONS_CycleStop) OTU(Robot.CMD) OTU(BarcodeScanner.CMD) OTU(Nest1Cylinder.CMD) OTU(Nest2Cylinder.CMD) OTU(LeakTester1.CMD) OTU(LeakTester2.CMD) OTU(Conveyor.CMD) OTU(RFIDScanner.CMD) ,MOVE(0,OP220_Seq.NextStep) MOVE(0,LeakTester1.Step[0]) MOVE(0,LeakTester2.Step[0]) ];
   18: [XIO(OP220.InCycle) MOVE(0,OP220.CycleStop_IND) ,XIC(OP220.InCycle) XIO(OP220.CycleStopRequested) MOVE(1,OP220.CycleStop_IND) ,XIC(PLC.AlwaysOff) MOVE(2,OP220.CycleStop_IND) ,XIC(OP220.InCycle) XIC(OP220.CycleStopRequested) MOVE(3,OP220.CycleStop_IND) ,XIC(PLC.AlwaysOff) MOVE(4,OP220.CycleStop_IND) ];
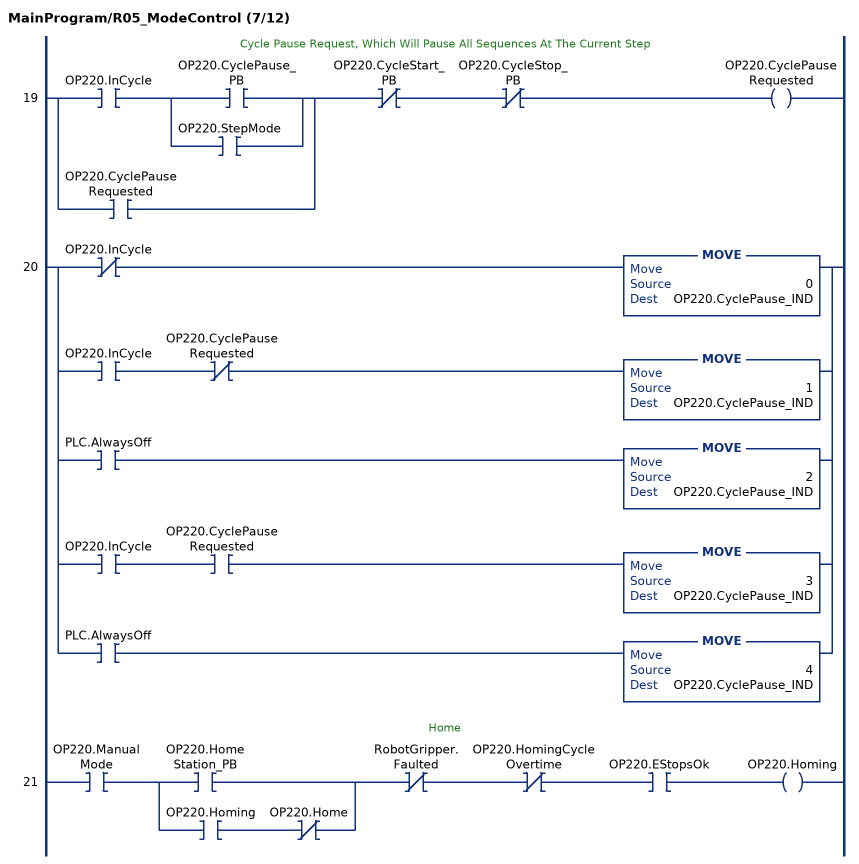
   // Cycle Pause Request, Which Will Pause All Sequences At The Current Step
   19: [XIC(OP220.InCycle) [XIC(OP220.CyclePause_PB) ,XIC(OP220.StepMode) ] ,XIC(OP220.CyclePauseRequested) ]XIO(OP220.CycleStart_PB)XIO(OP220.CycleStop_PB)OTE(OP220.CyclePauseRequested);
   20: [XIO(OP220.InCycle) MOVE(0,OP220.CyclePause_IND) ,XIC(OP220.InCycle) XIO(OP220.CyclePauseRequested) MOVE(1,OP220.CyclePause_IND) ,XIC(PLC.AlwaysOff) MOVE(2,OP220.CyclePause_IND) ,XIC(OP220.InCycle) XIC(OP220.CyclePauseRequested) MOVE(3,OP220.CyclePause_IND) ,XIC(PLC.AlwaysOff) MOVE(4,OP220.CyclePause_IND) ];
   // Home
   21: XIC(OP220.ManualMode)[XIC(OP220.HomeStation_PB) ,XIC(OP220.Homing) XIO(OP220.Home) ]XIO(RobotGripper.Faulted)XIO(OP220.HomingCycleOvertime)XIC(OP220.EStopsOk)OTE(OP220.Homing);
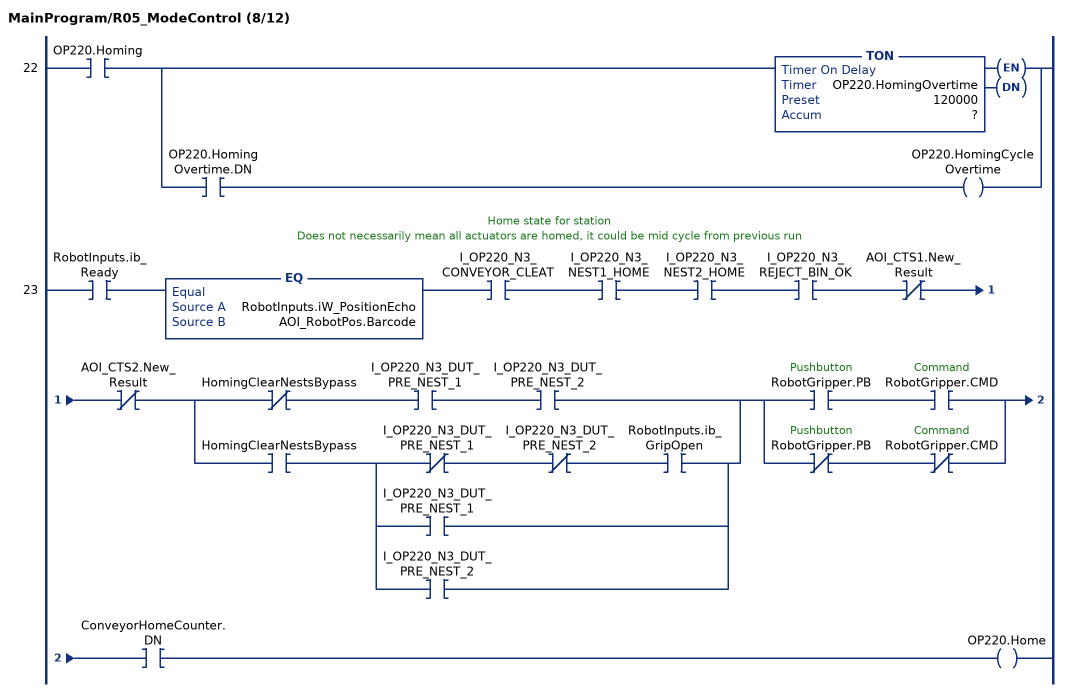
   22: XIC(OP220.Homing)[TON(OP220.HomingOvertime,?,?) ,XIC(OP220.HomingOvertime.DN) OTE(OP220.HomingCycleOvertime) ];
   // Home state for station
   // Does not necessarily mean all actuators are homed, it could be mid cycle from previous run
   23: XIC(RobotInputs.ib_Ready)EQ(RobotInputs.iW_PositionEcho,AOI_RobotPos.Barcode)XIC(I_OP220_N3_CONVEYOR_CLEAT)XIC(I_OP220_N3_NEST1_HOME)XIC(I_OP220_N3_NEST2_HOME)XIC(I_OP220_N3_REJECT_BIN_OK)XIO(AOI_CTS1.New_Result)XIO(AOI_CTS2.New_Result)[XIO(HomingClearNestsBypass) XIC(I_OP220_N3_DUT_PRE_NEST_1) XIC(I_OP220_N3_DUT_PRE_NEST_2) ,XIC(HomingClearNestsBypass) [XIO(I_OP220_N3_DUT_PRE_NEST_1) XIO(I_OP220_N3_DUT_PRE_NEST_2) XIC(RobotInputs.ib_GripOpen) ,XIC(I_OP220_N3_DUT_PRE_NEST_1) ,XIC(I_OP220_N3_DUT_PRE_NEST_2) ] ][XIC(RobotGripper.PB) XIC(RobotGripper.CMD) ,XIO(RobotGripper.PB) XIO(RobotGripper.CMD) ]XIC(ConveyorHomeCounter.DN)OTE(OP220.Home);
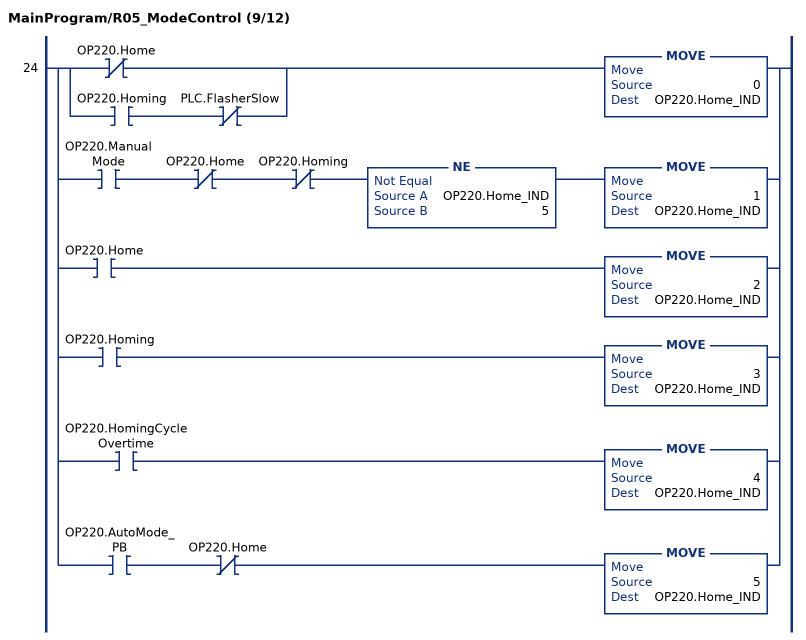
   24: [[XIO(OP220.Home) ,XIC(OP220.Homing) XIO(PLC.FlasherSlow) ] MOVE(0,OP220.Home_IND) ,XIC(OP220.ManualMode) XIO(OP220.Home) XIO(OP220.Homing) NE(OP220.Home_IND,5) MOVE(1,OP220.Home_IND) ,XIC(OP220.Home) MOVE(2,OP220.Home_IND) ,XIC(OP220.Homing) MOVE(3,OP220.Home_IND) ,XIC(OP220.HomingCycleOvertime) MOVE(4,OP220.Home_IND) ,XIC(OP220.AutoMode_PB) XIO(OP220.Home) MOVE(5,OP220.Home_IND) ];
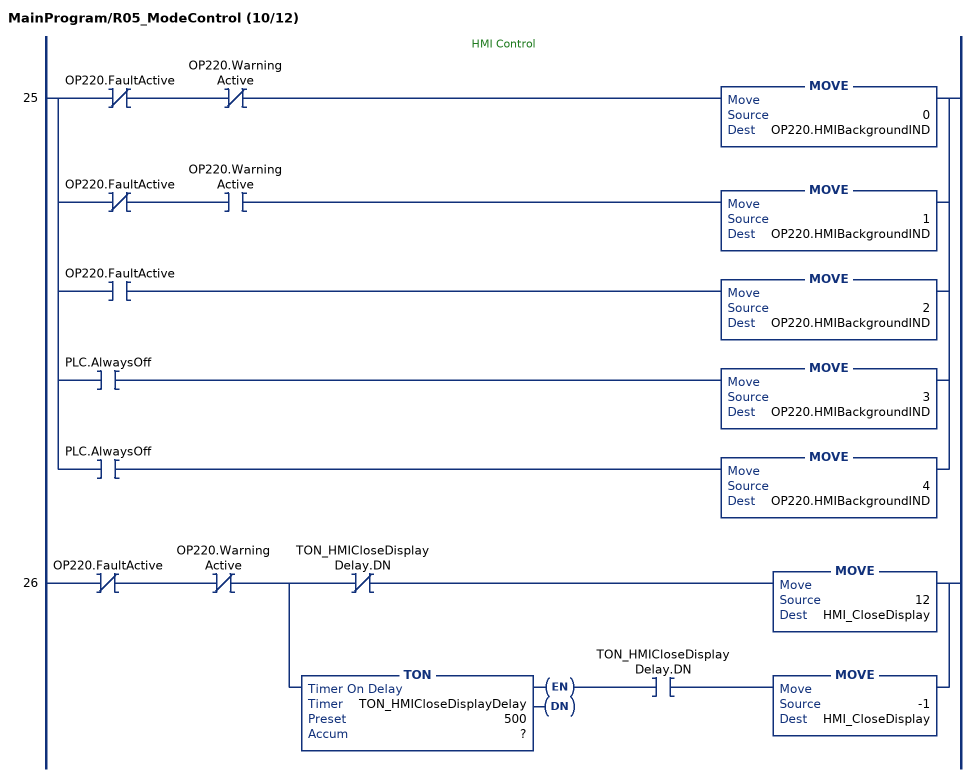
   // HMI Control
   25: [XIO(OP220.FaultActive) XIO(OP220.WarningActive) MOVE(0,OP220.HMIBackgroundIND) ,XIO(OP220.FaultActive) XIC(OP220.WarningActive) MOVE(1,OP220.HMIBackgroundIND) ,XIC(OP220.FaultActive) MOVE(2,OP220.HMIBackgroundIND) ,XIC(PLC.AlwaysOff) MOVE(3,OP220.HMIBackgroundIND) ,XIC(PLC.AlwaysOff) MOVE(4,OP220.HMIBackgroundIND) ];
   26: XIO(OP220.FaultActive)XIO(OP220.WarningActive)[XIO(TON_HMICloseDisplayDelay.DN) MOVE(12,HMI_CloseDisplay) ,TON(TON_HMICloseDisplayDelay,?,?) XIC(TON_HMICloseDisplayDelay.DN) MOVE(-1,HMI_CloseDisplay) ];
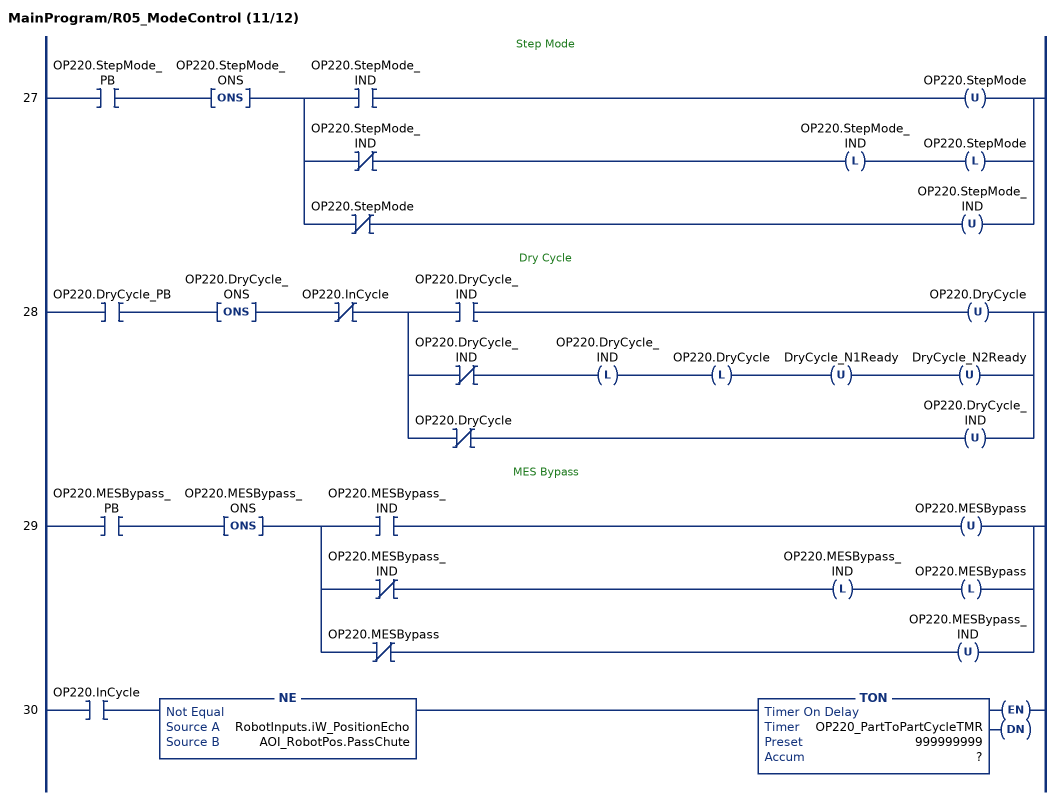
   // Step Mode
   27: XIC(OP220.StepMode_PB)ONS(OP220.StepMode_ONS)[XIC(OP220.StepMode_IND) OTU(OP220.StepMode) ,XIO(OP220.StepMode_IND) OTL(OP220.StepMode_IND) OTL(OP220.StepMode) ,XIO(OP220.StepMode) OTU(OP220.StepMode_IND) ];
   // Dry Cycle
   28: XIC(OP220.DryCycle_PB)ONS(OP220.DryCycle_ONS)XIO(OP220.InCycle)[XIC(OP220.DryCycle_IND) OTU(OP220.DryCycle) ,XIO(OP220.DryCycle_IND) OTL(OP220.DryCycle_IND) OTL(OP220.DryCycle) OTU(DryCycle_N1Ready) OTU(DryCycle_N2Ready) ,XIO(OP220.DryCycle) OTU(OP220.DryCycle_IND) ];
   // MES Bypass
   29: XIC(OP220.MESBypass_PB)ONS(OP220.MESBypass_ONS)[XIC(OP220.MESBypass_IND) OTU(OP220.MESBypass) ,XIO(OP220.MESBypass_IND) OTL(OP220.MESBypass_IND) OTL(OP220.MESBypass) ,XIO(OP220.MESBypass) OTU(OP220.MESBypass_IND) ];
   30: XIC(OP220.InCycle)NE(RobotInputs.iW_PositionEcho,AOI_RobotPos.PassChute)TON(OP220_PartToPartCycleTMR,?,?);
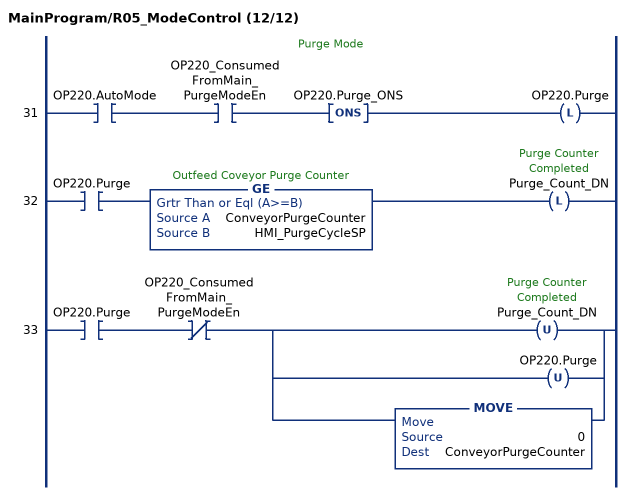
   // Purge Mode
   31: XIC(OP220.AutoMode)XIC(OP220_ConsumedFromMain_PurgeModeEn)ONS(OP220.Purge_ONS)OTL(OP220.Purge);
   32: XIC(OP220.Purge)GE(ConveyorPurgeCounter,HMI_PurgeCycleSP)OTL(Purge_Count_DN);
   33: XIC(OP220.Purge)XIO(OP220_ConsumedFromMain_PurgeModeEn)[OTU(Purge_Count_DN) ,OTU(OP220.Purge) ,MOVE(0,ConveyorPurgeCounter) ];
END_ROUTINE
